Universal Robots PolyScope program: new_piece_setup.urp

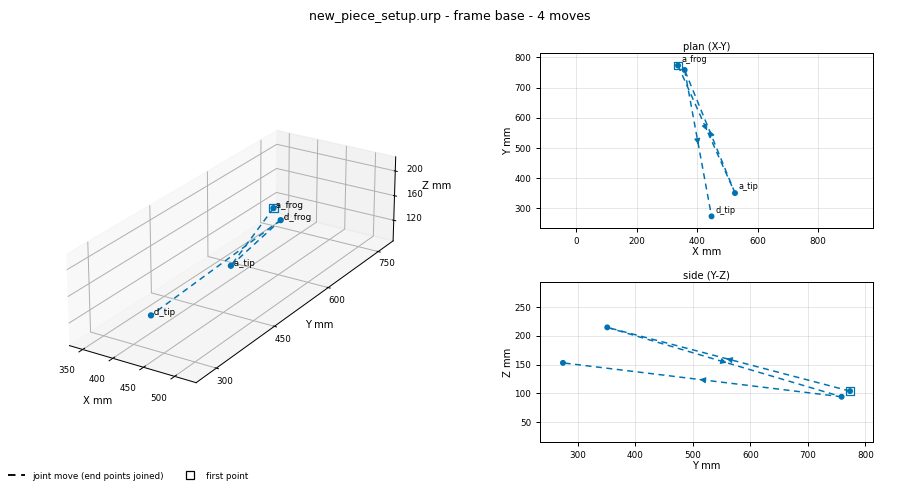
[picture p0: tool path of new_piece_setup.urp in frame base, 4 of 4 moves have a stored position in this frame; points joined in program order, loops and branches not executed]
Program new_piece_setup (installation=string_planes directory=/programs/hard_coded_pieces createdIn=5.17.3 lastSavedIn=5.17.3 robotSerialNumber=20245501435)
Calibrated DH parameters: a=[0.000154, -0.137004, -0.385524, -0.00002, 0.000092, 0]; d=[0.162441, 211.794786, -230.585024, 18.923638, 0.099786, 0.09951]; alpha=[1.569493, -0.001902, 0.003874, 1.570111, -1.570167, 0]; deltaTheta=[0, -1.242934, 1.056292, 0.186646, 0.000002, 0.000001]
InitVariablesNode
Robot Program (runOnlyOnce=false)
  MoveJ speed 60 deg/s, acceleration 80 deg/s^2 (useActiveTCP=true) feature=Base
    Waypoint a_frog: TCP in base x=336.638 y=773.336 z=103.937 mm, rx=-1.3698 ry=-2.3362 rz=1.327 rad; joints [-127.102, -6.181, 18.995, -50.118, -88.699, -156.884] deg; TCP offset x=28.21 y=-96.107 z=-99.69 mm, rx=0 ry=0 rz=0 rad
    Waypoint a_tip: TCP in base x=525.206 y=350.983 z=214.78 mm, rx=-1.3698 ry=-2.3362 rz=1.327 rad; joints [-161.028, -44.56, 81.191, -78.693, -115.03, -178.818] deg
    Waypoint d_frog: TCP in base x=358.556 y=758.659 z=94.067 mm, rx=-1.5094 ry=-2.0788 rz=1.1993 rad; joints [-129.115, -10.524, 30.67, -58.491, -76.391, -153.642] deg
    Waypoint d_tip: TCP in base x=447.609 y=273.936 z=153.016 mm, rx=-1.5094 ry=-2.0788 rz=1.1993 rad; joints [-166.924, -49.251, 104.272, -93.996, -106.227, -176.948] deg
